// TIA Portal V18 export
TYPE "typePOSMEMcalib"
// stored: IsFailsafeCompliant false
   STRUCT
      MEM : Real;
      offset : Real;
      calibrated : Bool;
   END_STRUCT;
END_TYPE
